PROPERTY IdentifiedBTN : STRING
GET
IF ipMoverTcIo <> 0 THEN
	_IdentifiedBTN := ipMoverTcIo.GetIdentifiedMoverBtn();
END_IF

IdentifiedBTN := _IdentifiedBTN;
END_GET
SET
_IdentifiedBTN := IdentifiedBTN;
END_SET
END_PROPERTY

PROPERTY InStation : BOOL
GET
InStation := _InStation;
END_GET
SET
_InStation := InStation;
END_SET
END_PROPERTY

METHOD LeaveMovementArea : I_PlanarTaskResult
LeaveMovementArea := LeaveMvmtAreaTask.Execute();
END_METHOD

PROPERTY MoveCommand : I_MoveCommands
GET
MoveCommand := THIS^;
END_GET
END_PROPERTY

PROPERTY MoverBTN : STRING
GET
IF ipMoverTcIo <> 0 THEN
	_MoverBTN := ipMoverTcIo.GetBtn();
END_IF

MoverBTN := _MoverBTN;
END_GET
END_PROPERTY

PROPERTY MoverIndex : UDINT
GET
MoverIndex := _MoverIndex;
END_GET
SET
_MoverIndex := MoverIndex;
END_SET
END_PROPERTY

PROPERTY MoverType : XPlanarMoverType
GET
MoverType := _MoverType;
END_GET
SET
_MoverType := MoverType;
END_SET
END_PROPERTY

PROPERTY ObjectInfo : REFERENCE TO PlanarObjectInfo
GET
ObjectInfo ref= _ObjectInfo;
END_GET
END_PROPERTY

{attribute 'suppress_wrn_C0410'}
PROPERTY pm : REFERENCE TO MC_PlanarMover
GET
pm ref= _Mover;
END_GET
END_PROPERTY

METHOD PUBLIC Reset : I_PlanarTaskResult
Reset := ResetMover.Execute();
END_METHOD

PROPERTY RotationModulo : LREAL
GET
RotationModulo := _ModuloPosC;
END_GET
END_PROPERTY

{attribute 'suppress_wrn_C0410'}
PROPERTY Status : REFERENCE TO CDT_MCTOPLC_PLANAR_MOVER_STD
GET
Status ref= _Std;
END_GET
END_PROPERTY

PROPERTY Utility : I_TcIoXPlanarMover
GET
IF ipMoverTcIo <> 0 THEN
	Utility := ipMoverTcIo;
END_IF
END_GET
SET
ipMoverTcIo := Utility;
END_SET
END_PROPERTY

METHOD CyclicLogic
VAR
	Result : BOOL;
END_VAR

VAR_INST
	MoverSetPos	 : MoverVector;
	SetPosX		 : LREAL;
	SetPosY		 : LREAL;
	ModXPos		 : LREAL;
	ModXPosRound : LREAL;
	ModYPos		 : LREAL;
	ModYPosRound : LREAL;
	FracX		 : LREAL;
	FracY		 : LREAL;
END_VAR
//Keep Task command feedbacks up to date
EnableMover.CyclicLogic();
DisableMover.CyclicLogic();
HaltMover.CyclicLogic();
JoinMoverToTrack.CyclicLogic();
LeaveMoverFromTrack.CyclicLogic();
ResetMover.CyclicLogic();
MoveOnTrackXY.CyclicLogic();
MoveOnTrack.CyclicLogic();
RotateMover.CyclicLogic();
XMove.CyclicLogic();
YMove.CyclicLogic();
ZMove.CyclicLogic();
AMove.CyclicLogic();
BMove.CyclicLogic();
XMoveRelative.CyclicLogic();
YMoveRelative.CyclicLogic();
CMoveRelative.CyclicLogic();
XMoveVelocity.CyclicLogic();
YMoveVelocity.CyclicLogic();
CMoveVelocity.CyclicLogic();
MoveToPosition.CyclicLogic();
AddMoverToGroup.CyclicLogic();
JoinToClosestTrack.CyclicLogic();
SquareMover.CyclicLogic();
RunExternalSetpointRelativeMode.CyclicLogic();
StopExternalSetpoint.CyclicLogic();
EnterMvmtAreaTask.CyclicLogic();
LeaveMvmtAreaTask.CyclicLogic();

IF NOT _Initialized THEN
	RETURN;
END_IF

//Update Mover MC Info
_std	 := _Mover.MCTOPLC.STD;
_Busy	 := _std.Busy.busyMover;
_Error	 := _Mover.Error;
_ErrorID := _Mover.ErrorId;

//Get Current Mover Position
_PreviousActPos := _MoverActPos;
_MoverActPos := _Mover.MCTOPLC.ACT.ActPos;

//Calculate Mover Closest Quarter Angle
_ModuloPosC	 := MODABS(_MoverActPos.c, 360.0);
IF _ModuloPosC < 315.0 AND _ModuloPosC > 225.0 THEN
	_ClosestQuarterAngle := 270.0;
ELSIF _ModuloPosC < 225.0 AND _ModuloPosC > 135.0 THEN
	_ClosestQuarterAngle := 180.0;
ELSIF _ModuloPosC < 135.0 AND _ModuloPosC > 45.0 THEN
	_ClosestQuarterAngle := 90.0;
ELSE
	_ClosestQuarterAngle := 0.0;
END_IF

//Determine if Mover is at a valid rotation position
MoverSetPos			:= _Mover.MCTOPLC.SET.SetPos;
SetPosX				:= TO_LREAL(TO_DINT(MoverSetPos.x * (2 * 10))) / (2 * 10); //Round the X position to 2 decimal places
SetPosY				:= TO_LREAL(TO_DINT(MoverSetPos.y * (2 * 10))) / (2 * 10); //Round the X position to 2 decimal places
ModXPos				:= LMOD(MoverSetPos.x, XPlanar.RotationMultiplier);
ModXPosRound		:= TO_LREAL(TO_DINT(ModXPos * (2 * 10))) / (2 * 10); //Round the Modulo position to 2 decimal places
FracX				:= FRAC(ModXPosRound);
ModYPos				:= LMOD(MoverSetPos.y, XPlanar.RotationMultiplier);
ModYPosRound		:= TO_LREAL(TO_DINT(ModYPos * (2 * 10))) / (2 * 10); //Round the Modulo position to 2 decimal places
FracY				:= FRAC(ModYPosRound);

//If APS42xx tiles are detected allow rotation anywhere on driver version 5 and above
IF Tc3_XPlanarUtility.Global_Version.stLibVersion_Tc3_XPlanarUtility.iMajor >= 5 AND XPlanar.RotationMultiplier = 80  THEN
	_AtRotationPosition := TRUE;
ELSE
	_AtRotationPosition := (SetPosX >= (XPlanar.RotationMultiplier - 0.25) AND FracX = 0) AND (SetPosY >= (XPlanar.RotationMultiplier - 0.25) AND FracY = 0);
END_IF

//Monitor Changes in move dynamic settings
IF UpdateMoveDynamics THEN
	_DynMove.SetValuesVADJ(_MoveDynamics.Velocity,
						   _MoveDynamics.Accel,
						   _MoveDynamics.Decel,
						   _MoveDynamics.Jerk);

	_DynTrackMove.SetValuesVADJ(_MoveDynamics.Velocity,
								_MoveDynamics.Accel,
								_MoveDynamics.Decel,
								_MoveDynamics.Jerk);

	UpdateMoveDynamics := FALSE;
END_IF

IF UpdateRotateDynamics THEN
	_DynRotate.SetLimit(Coord_Mcs_C1,
						_RotateDynamics.Velocity,
						_RotateDynamics.Accel,
						_RotateDynamics.Decel,
						_RotateDynamics.Jerk);

	UpdateRotateDynamics := FALSE;
END_IF

IF UpdateTiltDynamics THEN
	_DynRotate.SetLimit(Coord_Mcs_A1,
						_TiltDynamics.Velocity,
						_TiltDynamics.Accel,
						_TiltDynamics.Decel,
						_TiltDynamics.Jerk);

	_DynRotate.SetLimit(Coord_Mcs_B1,
						_TiltDynamics.Velocity,
						_TiltDynamics.Accel,
						_TiltDynamics.Decel,
						_TiltDynamics.Jerk);

	UpdateTiltDynamics := FALSE;
END_IF

//Update Mover Position for HMI
IF _MoverIndex > 0 AND _MoverIndex <= HmiObjectCounts.Movers THEN
	XPlanarHMI.MoverPositions[_MoverIndex]		  := _MoverActPos;
	XPlanarHMI.MoverObjects[_MoverIndex].MoverBTN := _MoverBTN;
	XPlanarHMI.MoverObjects[_MoverIndex].Error	  := _Error;
END_IF
END_METHOD

//FB_Init is always available implicitly and it is used primarily for initialization.
//The return value is not evaluated. For a specific influence, you can also declare the
//methods explicitly and provide additional code there with the standard initialization
//code. You can evaluate the return value.
METHOD FB_Init: BOOL
VAR_INPUT
    bInitRetains: BOOL; // TRUE: the retain variables are initialized (reset warm / reset cold)
    bInCopyCode: BOOL;  // TRUE: the instance will be copied to the copy code afterward (online change)   
END_VAR
VAR
	i	: UINT;
END_VAR
IF NOT bInCopyCode THEN
	FOR i := 1 TO Tc3_XPlanarUtility.Param_TcIoXPlanarEnvironment.MaxMcPlanarMovers DO
		IF ip.Movers[i] = 0 THEN
			ip.Movers[i] := THIS^;
			ip.Movers[i].MoverIndex := i;
			EXIT;
		END_IF 
	END_FOR
END_IF
END_METHOD

PROPERTY LastCyclePosition : Reference TO MoverVector
GET
LastCyclePosition ref= _PreviousActPos;
END_GET
END_PROPERTY

PROPERTY MoverData : I_MoverData
GET
MoverData := _MoverData;
END_GET
SET
_MoverData := MoverData;
END_SET
END_PROPERTY

END_FUNCTION_BLOCK

// Part/Tasks/FB_AllowEnable
FUNCTION_BLOCK FB_AllowEnable EXTENDS FB_PartTask
VAR
END_VAR

METHOD Execute : I_PlanarTaskResult
VAR_INPUT
END_VAR
IF NOT HasRun THEN
	_Done	 := FALSE;
	_Error	 := FALSE;
	_Busy	 := FALSE;
	_ErrorID := 0;
	ipPart.pm.AllowEnable(_PlanarFb);
	HasRun := TRUE;
END_IF

Execute := THIS^;

//Heartbeat that the method is active
ExecuteWatchdog := ExecuteWatchdog + 1;
END_METHOD

END_FUNCTION_BLOCK

// Part/Tasks/FB_ForceDisable
FUNCTION_BLOCK FB_ForceDisable EXTENDS FB_PartTask
VAR
END_VAR

METHOD Execute : I_PlanarTaskResult
VAR_INPUT
END_VAR
IF NOT HasRun THEN
	_Done	 := FALSE;
	_Error	 := FALSE;
	_Busy	 := FALSE;
	_ErrorID := 0;
	ipPart.pm.ForceDisable(_PlanarFb);
	HasRun := TRUE;
END_IF

Execute := THIS^;

//Heartbeat that the method is active
ExecuteWatchdog := ExecuteWatchdog + 1;
END_METHOD

END_FUNCTION_BLOCK

// Part/Tasks/FB_Initialize
FUNCTION_BLOCK FB_Initialize EXTENDS FB_PartTask
VAR
END_VAR

METHOD Execute : I_PlanarTaskResult
VAR_INPUT
	OID : OTCID;
END_VAR
IF NOT HasRun THEN
	ipPart.pm.Initialize(_PlanarFb, OID, XPlanar.Environment);
	HasRun := TRUE;
END_IF

Execute := THIS^;

//Heartbeat that the method is active
ExecuteWatchdog := ExecuteWatchdog + 1;
END_METHOD

END_FUNCTION_BLOCK

// Part/Tasks/FB_ResetPart
FUNCTION_BLOCK FB_ResetPart EXTENDS FB_PartTask
VAR
END_VAR

METHOD Execute : I_PlanarTaskResult
VAR_INPUT
END_VAR
IF NOT HasRun THEN
	_Done	 := FALSE;
	_Error	 := FALSE;
	_Busy	 := FALSE;
	_ErrorID := 0;
	ipPart.pm.Reset(_PlanarFb);
	HasRun := TRUE;
END_IF

Execute := THIS^;

//Heartbeat that the method is active
ExecuteWatchdog := ExecuteWatchdog + 1;
END_METHOD

END_FUNCTION_BLOCK

// Part/FB_XPlanarPart
{attribute 'no_assign'}
{attribute 'no_explicit_call' := 'do not call this POU directly'}
FUNCTION_BLOCK FB_XPlanarPart IMPLEMENTS I_XPlanarPart
VAR
	{attribute 'suppress_wrn_C0540'}
	PlanarPart			 : MC_PlanarPart;
	_Busy				 : BOOL;
	_Error				 : BOOL;
	_ErrorID			 : UDINT;
	_ObjectID			 : OTCID;
	InitPart			 : FB_Initialize   := (Part := THIS^);
	AllowPartEnable		 : FB_AllowEnable  := (Part := THIS^);
	ForcePartDisable	 : FB_ForceDisable := (Part := THIS^);
	ResetPart			 : FB_ResetPart	   := (Part := THIS^);
	InvalidCommandResult : FB_TaskResult   := (Busy := FALSE, Error := TRUE, ErrorID := 9999);
END_VAR

PROPERTY Busy : BOOL
GET
Busy := _Busy;
END_GET
END_PROPERTY

METHOD PUBLIC CyclicLogic
VAR_INPUT
END_VAR
InitPart.CyclicLogic();
AllowPartEnable.CyclicLogic();
ForcePartDisable.CyclicLogic();
ResetPart.CyclicLogic();
END_METHOD

PROPERTY Error : BOOL
GET
Error := _Error;
END_GET
END_PROPERTY

PROPERTY ErrorId : UDINT
GET
ErrorId := ErrorID;
END_GET
END_PROPERTY

METHOD ForceDisable : I_PlanarTaskResult
ForceDisable := ForcePartDisable.Execute();
END_METHOD

METHOD Initialize : I_PlanarTaskResult
VAR_INPUT
END_VAR
IF _ObjectID <> 0 THEN
	Initialize := InitPart.Execute(_ObjectID);
ELSE
	Initialize := InvalidCommandResult;
END_IF
END_METHOD

PROPERTY ObjectID : OTCID
GET
ObjectID := _ObjectID;
END_GET
SET
_ObjectID := ObjectID;
END_SET
END_PROPERTY

{attribute 'suppress_wrn_C0410'}
PROPERTY pm : REFERENCE TO MC_PlanarPart
GET
pm  ref= PlanarPart;
END_GET
END_PROPERTY

METHOD Reset : I_PlanarTaskResult
VAR_INPUT
END_VAR
Reset := ResetPart.Execute();
END_METHOD

METHOD SetAllowEnable : I_PlanarTaskResult
SetAllowEnable := AllowPartEnable.Execute();
END_METHOD

{attribute 'suppress_wrn_C0410'}
PROPERTY State : REFERENCE TO MC_PLANAR_STATE
GET
State := PlanarPart.State;
END_GET
END_PROPERTY

END_FUNCTION_BLOCK

// PositionTrigger/FB_XPlanarPositionTrigger
FUNCTION_BLOCK FB_XPlanarPositionTrigger IMPLEMENTS I_Cyclic, I_XPlanarPositionTrigger
VAR
	_Position		  : FB_PositionXY;
	_Queue			  : FB_MoverQueue;
	_RegisteredMovers : FB_MoverList;
	AllMovers		  : BOOL;
END_VAR

METHOD CyclicLogic
WatchForMover();
END_METHOD

METHOD DeregisterMover
VAR_INPUT
	Mover	: I_XPlanarMover;
END_VAR
_RegisteredMovers.RemoveMover(Mover);
END_METHOD

METHOD GetMover : I_XPlanarMover
GetMover := _Queue.Dequeue();
END_METHOD

PROPERTY MoverIsPresent : BOOL
GET
MoverIsPresent := _Queue.Count > 0;
END_GET
END_PROPERTY

PROPERTY MoverQueue : I_MoverQueue
GET
MoverQueue := _Queue;
END_GET
END_PROPERTY

PROPERTY Position : I_HasPosition
GET
Position := _Position;
END_GET
END_PROPERTY

METHOD RegisterAllMovers
AllMovers := TRUE;
END_METHOD

METHOD RegisterMover
VAR_INPUT
	Mover	: I_XPlanarMover;
END_VAR
VAR
	i : UDINT;
END_VAR
FOR i := 1 TO _RegisteredMovers.Count DO
	IF _RegisteredMovers.List[i] = Mover THEN
		RETURN;
	END_IF
END_FOR
_RegisteredMovers.AddMover(Mover);
END_METHOD

METHOD WatchForMover
VAR_INST
	i : UDINT;
END_VAR

VAR
	idx: UDINT;
END_VAR
IF AllMovers THEN
	FOR i := 1 TO XPlanar.MoverCount DO
		IF ip.Movers[i] <> 0 AND_THEN _Position.x > 0 AND _Position.y > 0 THEN
			IF (ip.Movers[i].ActualPosition.x >= _Position.x - 10 AND ip.Movers[i].ActualPosition.x <= _Position.x + 10) THEN 		//Paint the window in X
				IF _Position.y >= ip.Movers[i].LastCyclePosition.y AND _Position.y <= ip.Movers[i].ActualPosition.y OR 				//Wach for threshold in Y	
					_Position.y <= ip.Movers[i].LastCyclePosition.y AND _Position.y >= ip.Movers[i].ActualPosition.y THEN
						_Queue.Enqueue(ip.Movers[i]);
				END_IF
			ELSIF (ip.Movers[i].ActualPosition.y >= _Position.y - 10 AND ip.Movers[i].ActualPosition.y <= _Position.y + 10) THEN	//Paint the window in Y
				IF _Position.x >= ip.Movers[i].LastCyclePosition.x AND _Position.x <= ip.Movers[i].ActualPosition.x OR				//Wach for threshold in X
					_Position.x <= ip.Movers[i].LastCyclePosition.x AND _Position.x >= ip.Movers[i].ActualPosition.x THEN
						_Queue.Enqueue(ip.Movers[i]);
				END_IF
			END_IF
		END_IF
	END_FOR
ELSE
	FOR i := 1 TO _RegisteredMovers.Count DO
		IF _RegisteredMovers.List[i] <> 0 AND_THEN _Position.x > 0 AND _Position.y > 0 THEN
			IF (_RegisteredMovers.List[i].ActualPosition.x >= _Position.x - 10 AND _RegisteredMovers.List[i].ActualPosition.x <= _Position.x + 10) THEN 		//Paint the window in X
				IF _Position.y >= _RegisteredMovers.List[i].LastCyclePosition.y AND _Position.y <= _RegisteredMovers.List[i].ActualPosition.y OR 				//Wach for threshold in Y	
					_Position.y <= _RegisteredMovers.List[i].LastCyclePosition.y AND _Position.y >= _RegisteredMovers.List[i].ActualPosition.y THEN
						_Queue.Enqueue(_RegisteredMovers.List[i]);
				END_IF
			ELSIF (_RegisteredMovers.List[i].ActualPosition.y >= _Position.y - 10 AND _RegisteredMovers.List[i].ActualPosition.y <= _Position.y + 10) THEN		//Paint the window in Y
				IF _Position.x >= _RegisteredMovers.List[i].LastCyclePosition.x AND _Position.x <= _RegisteredMovers.List[i].ActualPosition.x OR				//Wach for threshold in X
					_Position.x <= _RegisteredMovers.List[i].LastCyclePosition.x AND _Position.x >= _RegisteredMovers.List[i].ActualPosition.x THEN
						_Queue.Enqueue(_RegisteredMovers.List[i]);
				END_IF
			END_IF
		END_IF
	END_FOR	
END_IF
END_METHOD

END_FUNCTION_BLOCK

// PositionTrigger/I_XPlanarPositionTrigger
INTERFACE I_XPlanarPositionTrigger EXTENDS I_Cyclic

METHOD DeregisterMover
VAR_INPUT
	Mover	: I_XPlanarMover;
END_VAR
END_METHOD

METHOD GetMover : I_XPlanarMover
END_METHOD

PROPERTY MoverIsPresent : BOOL
GET
END_GET
END_PROPERTY

PROPERTY MoverQueue : I_MoverQueue
GET
END_GET
END_PROPERTY

PROPERTY Position : I_HasPosition
GET
END_GET
END_PROPERTY

METHOD RegisterAllMovers
END_METHOD

METHOD RegisterMover
VAR_INPUT
	Mover	: I_XPlanarMover;
END_VAR
END_METHOD

END_INTERFACE

// Project Information/F_GetCompany
// This function has been automatically generated from the project information.
{attribute 'signature_flag' := '1073741824'}
{attribute 'TcGenerated'}
{attribute 'no-analysis'}
FUNCTION F_GetCompany : WSTRING
VAR_INPUT
	
END_VAR

F_GetCompany := "Beckhoff Automation LLC";

END_FUNCTION

// Project Information/F_GetTitle
// This function has been automatically generated from the project information.
{attribute 'signature_flag' := '1073741824'}
{attribute 'TcGenerated'}
{attribute 'no-analysis'}
FUNCTION F_GetTitle : WSTRING
VAR_INPUT
	
END_VAR

F_GetTitle := "XPlanarApplication";

END_FUNCTION

// Project Information/F_GetVersion
// This function has been automatically generated from the project information.
{attribute 'signature_flag' := '1073741824'}
{attribute 'TcGenerated'}
{attribute 'no-analysis'}
FUNCTION F_GetVersion : ST_LibVersion
VAR_INPUT
	
END_VAR

F_GetVersion.iMajor := 2;
F_GetVersion.iMinor := 0;
F_GetVersion.iBuild := 6;
F_GetVersion.iRevision := 0;
F_GetVersion.sVersion := '2.0.6';
F_GetVersion.nFlags := 0;

END_FUNCTION

// Station/FB_XPlanarStationBase
{attribute 'no_assign_warning'}
{attribute 'no_explicit_call' := 'do not call this POU directly'}
FUNCTION_BLOCK FB_XPlanarStationBase IMPLEMENTS I_Cyclic, I_XPlanarStation
VAR
	_Name				 : STRING;
	_Busy				 : BOOL;
	_Error				 : BOOL;
	_ErrorID			 : UDINT;
	_Position			 : PositionXYC; //Position of center of the zone
	ipCurrentMover		 : I_XPlanarMover;
	_MoverList			 : FB_MoverList;
	_NumMoversRequired	 : UDINT := 1;
	_ID					 : UDINT;
	_Size				 : Position2D_LREAL := (x := 50, y := 50); //Size of station in mm
	_HasMover			 : BOOL;
	_Occupied			 : BOOL;
	ipTrackID			 : UDINT;		 //ID of track that zone resides on
	_CanReleaseMover	 : BOOL := TRUE; //Set to 0 if station area is blocked
	_StationReady AT %Q* : BOOL;
	ipNextStation		 : I_XPlanarStation;
	_AllowQueing		 : BOOL := TRUE;
	_StationComplete	 : BOOL;
	_StationType		 : E_StationType := E_StationType.Process;
	PrepState			 : UDINT;
	StationState		 : E_XplanarStationState;
	i					 : UDINT := 1;
	CommandResult		 : I_PlanarTaskResult;
	_Process			 : I_StationProcess;
END_VAR

PROPERTY Process : I_StationProcess
GET
IF _Process <> 0 THEN
	Process := _Process;
END_IF
END_GET
SET
_Process := Process;
END_SET
END_PROPERTY

PROPERTY AllowQueing : BOOL
GET
AllowQueing := _AllowQueing;
END_GET
SET
_AllowQueing := AllowQueing;
END_SET
END_PROPERTY

PROPERTY CanReleaseMover : BOOL
SET
_CanReleaseMover := CanReleaseMover;
END_SET
END_PROPERTY

PROPERTY CurrentMover : I_XPlanarMover
GET
IF ipCurrentMover <> 0 THEN
	CurrentMover := ipCurrentMover;
END_IF
END_GET
END_PROPERTY

PROPERTY Error : BOOL
GET
Error := _Error;
END_GET
END_PROPERTY

METHOD Execute
WatchForMover();
IF ipCurrentMover <> 0 THEN
	CASE StationState OF
		E_XplanarStationState.StationIdle: //Wait for mover to arrive in position
			IF _HasMover AND _StationReady AND NOT _StationComplete THEN
				IF ipCurrentMover <> 0 THEN
					IF (ipTrackID <> 0 AND (ipCurrentMover.Status.CommandMode = MC_PLANAR_MOVER_COMMAND_MODE.OnTrack OR ipCurrentMover.Status.CommandMode = MC_PLANAR_MOVER_COMMAND_MODE.CRotationOnTrack)) OR (ipTrackID = 0 AND (ipCurrentMover.Status.CommandMode = MC_PLANAR_MOVER_COMMAND_MODE.FreeMovement OR ipCurrentMover.Status.CommandMode = MC_PLANAR_MOVER_COMMAND_MODE.CRotationFreeMovement))
						THEN
						StationState := E_XplanarStationState.ProcessMover;
					END_IF
				END_IF
			END_IF

		E_XplanarStationState.ProcessMover: //Perform the desired processes with the mover
			IF _Process <> 0 AND_THEN _Process.Execute(ipCurrentMover) THEN
				StationState := E_XplanarStationState.SquareUpMover;
			ELSIF _StationComplete THEN
				StationState := E_XplanarStationState.SquareUpMover;
			END_IF

		E_XplanarStationState.SquareUpMover: //Check mover for angle that allows X/Y Movement
			IF (ipCurrentMover.Status.CommandMode = MC_PLANAR_MOVER_COMMAND_MODE.CRotationOnTrack) OR (ipCurrentMover.Status.CommandMode = MC_PLANAR_MOVER_COMMAND_MODE.CRotationFreeMovement) THEN
				CommandResult := ipCurrentMover.MoveCommand.SquareUp();
				IF CommandResult.Done THEN
					StationState := E_XplanarStationState.SendMoverAway;
				END_IF
			ELSE
				StationState := E_XplanarStationState.SendMoverAway;
			END_IF

		E_XplanarStationState.SendMoverAway: //Send the current lead mover away
			IF ipNextStation <> 0 AND _CanReleaseMover THEN
				IF (NOT ipNextStation.HasMover OR ipNextStation.AllowQueing) THEN
					CommandResult := ipCurrentMover.MoveCommand.SendToStation(Destination := ipNextStation);
					IF CommandResult.Busy THEN
						StationState := E_XplanarStationState.CycleComplete;
					END_IF
				END_IF
			END_IF

		E_XplanarStationState.CycleComplete: //Mover on its way out
			_StationReady := FALSE;
			StationState  := E_XplanarStationState.StationIdle;

		E_XPlanarStationState.StationError:
			_Error := TRUE;
	END_CASE
ELSE
	_StationComplete := FALSE;
	_StationReady	 := FALSE;
	StationState	 := E_XplanarStationState.StationIdle;
END_IF
END_METHOD

PROPERTY HasMover : BOOL
GET
HasMover := _HasMover;
END_GET
SET
_HasMover := HasMover;
END_SET
END_PROPERTY

PROPERTY ID : UDINT
GET
ID := _ID;
END_GET
SET
_ID := ID;
END_SET
END_PROPERTY

{attribute 'suppress_wrn_C0410'}
PROPERTY MoverList : REFERENCE TO FB_MoverList
GET
MoverList ref= _MoverList;
END_GET
END_PROPERTY

PROPERTY NextStation : I_XPlanarStation
GET
NextStation := ipNextStation;
END_GET
SET
ipNextStation := NextStation;
END_SET
END_PROPERTY

{attribute 'suppress_wrn_C0410'}
PROPERTY Position : REFERENCE TO PositionXYC
GET
Position ref= _Position;
END_GET
END_PROPERTY

METHOD Reset : BOOL
StationState := E_XplanarStationState.StationIdle;
PrepState	 := 0;
_Error		 := FALSE;
Reset		 := true;
END_METHOD

{attribute 'suppress_wrn_C0410'}
PROPERTY Size : REFERENCE TO Position2D_LREAL
GET
Size ref= _Size;
END_GET
END_PROPERTY

PROPERTY StationComplete : BOOL
SET
_StationComplete := StationComplete;
END_SET
END_PROPERTY

PROPERTY StationReady : BOOL
GET
StationReady := _StationReady;
END_GET
END_PROPERTY

PROPERTY StationType : E_StationType
GET
StationType := _StationType;
END_GET
SET
_StationType := StationType;
END_SET
END_PROPERTY

PROPERTY TrackID : UDINT
GET
TrackID := ipTrackID;
END_GET
SET
ipTrackID := TrackID;
END_SET
END_PROPERTY

METHOD CyclicLogic
VAR
	i : UDINT;
END_VAR
IF _ID > 0 AND _ID <= XPlanar.StationCount THEN
	XPlanarHMI.StationObjects[_ID].Width  := TO_DINT(_Size.x);
	XPlanarHMI.StationObjects[_ID].Height := TO_DINT(_Size.y);
	XPlanarHMI.StationObjects[_ID].X	  := TO_DINT(_Position.x);
	XPlanarHMI.StationObjects[_ID].Y	  := TO_DINT(_Position.y);
END_IF

_Busy := _HasMover;

//Create a queue of all movers destined for this station
_MoverList.Clear();
FOR i := 1 TO XPlanar.MoverCount DO
	IF ip.Movers[i] <> 0 AND ip.Movers[i].Destination <> 0 THEN
		IF ip.Movers[i].Destination.ID = _ID THEN
			_MoverList.AddMover(ip.Movers[i]);
		END_IF
	END_IF
END_FOR
END_METHOD

//FB_Init is always available implicitly and it is used primarily for initialization.

//The return value is not evaluated. For a specific influence, you can also declare the

//methods explicitly and provide additional code there with the standard initialization

//code. You can evaluate the return value.
METHOD FB_Init : BOOL
VAR_INPUT
	bInitRetains : BOOL; // TRUE: the retain variables are initialized (reset warm / reset cold)
	bInCopyCode	 : BOOL; // TRUE: the instance will be copied to the copy code afterward (online change)   
END_VAR

VAR
	i : UINT;
END_VAR
IF NOT bInCopyCode THEN
	FOR i := 1 TO SystemParameters.MAX_STATION_COUNT DO
		IF ip.Stations[i] = 0 THEN
			ip.Stations[i] := THIS^;
			ip.Stations[i].ID := i;
			XPlanar.StationCount := i;
			EXIT;
		END_IF
	END_FOR
END_IF
END_METHOD

PROPERTY Name : STRING
GET
Name := _Name;
END_GET
SET
_Name := Name;
END_SET
END_PROPERTY

METHOD WatchForMover
VAR_INST
	idx : UDINT;
END_VAR
FOR idx := 1 TO XPlanar.MoverCount DO
	IF ip.Movers[idx] <> 0 THEN
		IF _Position.x > 0 AND _Position.y > 0 THEN
			IF (ip.Movers[idx].ActualPosition.x + 50 >= _Position.x - (_Size.x / 2) AND ip.Movers[idx].ActualPosition.x - 50 <= _Position.x + (_Size.x / 2)) AND
			   (ip.Movers[idx].ActualPosition.y + 50 >= _Position.y - (_Size.y / 2) AND ip.Movers[idx].ActualPosition.y - 50 <= _Position.y + (_Size.y / 2)) THEN
				IF ip.Movers[idx].Destination <> 0 THEN
					IF ip.Movers[idx].Destination.ID = _ID THEN
						ipCurrentMover := ip.Movers[idx];
						_HasMover := TRUE;
						EXIT;
					ELSE
						ipCurrentMover := 0;
						_HasMover := FALSE;
					END_IF
				END_IF
			END_IF
		END_IF
	END_IF
END_FOR

IF _HasMover AND ipCurrentMover <> 0 THEN
	IF ipCurrentMover <> 0 THEN
		CASE _StationType OF
			E_StationType.Process:
				_StationReady := NOT ipCurrentMover.Status.Busy.busyMover;

			E_StationType.DecisionPoint:
				_StationReady := _HasMover;
		END_CASE
	END_IF
END_IF
END_METHOD

END_FUNCTION_BLOCK

// Tile/FB_XPlanarTile
{attribute 'no_assign'}
{attribute 'no_explicit_call' := 'do not call this POU directly'}
FUNCTION_BLOCK FB_XPlanarTile
VAR
	_Busy				: BOOL;
	_Error				: BOOL;
	_ErrorID			: UDINT;
	_Utility			: I_TcIoXPlanarTile;
	_Index				: UINT;
	_Part				: UINT := 1;
	_Btn				: STRING(13);
	_DcLinkVoltage		: UINT;
	_DcLinkOk			: BOOL;
	_TimeToShutdown		: LREAL;
	_ObservedPower		: LREAL;
	_OverLimitFactor	: LREAL;
	_DiagData			: POINTER TO ST_CoeDriveDiagData;
	_Position			: ST_TcIoTilePositionOnPart;
	_Temperatures		: ST_TileTemperatures;
	_TileType			: TileType;
	CoEUpdateTimer		: TON;
	CriticalUpdateTimer : TON;
	DiagDataResult		: ULINT;
END_VAR

PROPERTY Btn : STRING(13)
GET
Btn := _Btn;
END_GET
END_PROPERTY

PROPERTY Busy : BOOL
GET
Busy := _Busy;
END_GET
END_PROPERTY

METHOD PUBLIC CyclicLogic
VAR_INST
	UpdateTileData : BOOL;
	test   : DINT;
END_VAR
(*IF XPlanar.OperationMode = Tc3_XPlanarUtility.XPlanarOperationMode.Normal THEN
	IF SystemParameters.TileDiagUpdate > 0 THEN
		CoEUpdateTimer(IN := NOT UpdateTileData, PT := TO_TIME(SystemParameters.TileDiagUpdate) * 1000);
		IF CoEUpdateTimer.Q THEN
			UpdateTileData := TRUE;
		END_IF

		test := SIZEOF(_diagdata);

		//Update the tile diagnostic data
		IF UpdateTileData AND_THEN XPlanar.EnvironmentTcIo.TcIoXpu(1).TcIoTile(_Part, Index).CoE.DiagData.Update() THEN
			_DiagData := XPlanar.EnvironmentTcIo.TcIoXpu(1).TcIoTile(_Part, Index).CoE.DiagData.All;
			_DcLinkOk := XPlanar.EnvironmentTcIo.TcIoXpu(1).TcIoTile(_Part, Index).CoE.DiagData.DcLinkOk;
			UpdateTileData	  := FALSE;
		END_IF

		CriticalUpdateTimer(IN := NOT CriticalUpdateTimer.Q, PT := T#1S);
		IF CriticalUpdateTimer.Q THEN
			_TimeToShutdown	 := XPlanar.EnvironmentTcIo.TcIoXpu(1).TcIoTile(_Part, Index).GetTimeToShutdown();
			_ObservedPower	 := XPlanar.EnvironmentTcIo.TcIoXpu(1).TcIoTile(_Part, Index).GetObservedTilePower();
			_OverLimitFactor := XPlanar.EnvironmentTcIo.TcIoXpu(1).TcIoTile(_Part, Index).GetPowerOverLimitFactor();
		END_IF
	ELSE
		UpdateTileData := FALSE;
	END_IF
END_IF
*)
END_METHOD

PROPERTY DcLinkOk : BOOL
GET
DcLinkOk := _DcLinkOk;
END_GET
END_PROPERTY

PROPERTY Error : BOOL
GET
Error := _Error;
END_GET
END_PROPERTY

PROPERTY ErrorId : UDINT
GET
ErrorId := ErrorID;
END_GET
END_PROPERTY

PROPERTY Index : UINT
GET
Index := _Index;
END_GET
SET
_Index := Index;
END_SET
END_PROPERTY

METHOD Initialize : BOOL
//Get the Tile Type
_TileType := XPlanar.EnvironmentTcIo.TcIoXpu(1).TcIoTile(_Part, _Index).GetTileType();

//Get the configured position of the tile
_Position := XPlanar.EnvironmentTcIo.TcIoXpu(1).TcIoTile(_Part, _Index).TilePositionOnPart();

//Get BTN of tile
_Btn := XPlanar.EnvironmentTcIo.TcIoXpu(1).TcIoTile(_Part, _Index).GetBtn();

//Update the object array for HMI
IF _Index > 0 AND _Index <= HMIObjectCounts.Tiles THEN
	//Populate tile position
	XPlanarHMI.TileObjects[_Index].X := TO_DINT(_Position.X);
	XPlanarHMI.TileObjects[_Index].Y := TO_DINT(_Position.Y);
	//Populate tile type
	CASE _TileType OF
		TileType.APS4224_1000_0000:
			XPlanarHMI.TileObjects[_Index].Width  := 160;
			XPlanarHMI.TileObjects[_Index].Height := 320;
			XPlanar.RotationMultiplier			  := 80.0;	
	
		TileType.APS4242_1000_0000:
			XPlanarHMI.TileObjects[_Index].Width  := 320;
			XPlanarHMI.TileObjects[_Index].Height := 160;
			XPlanar.RotationMultiplier			  := 80.0;	
			
		TileType.APS4244_1000_0000:
			XPlanarHMI.TileObjects[_Index].Width  := 320;
			XPlanarHMI.TileObjects[_Index].Height := 320;
			XPlanar.RotationMultiplier			  := 80.0;
	
		TileType.APS4322_0000_0000:
			XPlanarHMI.TileObjects[_Index].Width  := 240;
			XPlanarHMI.TileObjects[_Index].Height := 240;
			XPlanar.RotationMultiplier			  := 120.0;
	
// 			//Get initial diagnostic data
// 			IF _Part > 0 AND _Index > 0 THEN
// 				//ipTileTcIo := XPlanar.EnvironmentTcIo.TcIoXpu(1).TcIoTile(_Part, Index).Aps4322;
// 				IF XPlanar.OperationMode = Tc3_XPlanarUtility.XPlanarOperationMode.Normal THEN
// 					IF XPlanar.EnvironmentTcIo.TcIoXpu(1).TcIoTile(_Part, _Index).Aps4322.CoE.DiagData.Update() THEN
// 						_DiagData := XPlanar.EnvironmentTcIo.TcIoXpu(1).TcIoTile(_Part, _Index).Aps4322.CoE.DiagData.All;
// 					END_IF
// 				END_IF
// 			END_IF
	END_CASE
END_IF
Initialize := TRUE;
END_METHOD

PROPERTY PartIndex : UINT
GET
PartIndex := _Part;
END_GET
SET
_Part := PartIndex;
END_SET
END_PROPERTY

{attribute 'suppress_wrn_C0410'}
PROPERTY PositionOnPart : REFERENCE TO ST_TcIoTilePositionOnPart
GET
PositionOnPart ref= _Position;
END_GET
END_PROPERTY

{attribute 'suppress_wrn_C0410'}
PROPERTY Temperatures : REFERENCE TO ST_TileTemperatures
GET
Temperatures ref= _Temperatures;
END_GET
END_PROPERTY

PROPERTY TimeToShutdown : LREAL
GET
TimeToShutdown := _TimeToShutdown;
END_GET
END_PROPERTY

METHOD Update
VAR_INPUT
END_VAR
// XPlanar.EnvironmentTcIo.TcIoXpu(1).TcIoTile(_Part, Index).CoE.DiagData.Update();
// _DiagData		 := XPlanar.EnvironmentTcIo.TcIoXpu(1).TcIoTile(_Part, Index).CoE.DiagData.All;
// _DcLinkOk		 := XPlanar.EnvironmentTcIo.TcIoXpu(1).TcIoTile(_Part, Index).CoE.DiagData.DcLinkOk;
// _TimeToShutdown	 := XPlanar.EnvironmentTcIo.TcIoXpu(1).TcIoTile(_Part, Index).GetTimeToShutdown();
// _ObservedPower	 := XPlanar.EnvironmentTcIo.TcIoXpu(1).TcIoTile(_Part, Index).GetObservedTilePower();
// _OverLimitFactor := XPlanar.EnvironmentTcIo.TcIoXpu(1).TcIoTile(_Part, Index).GetPowerOverLimitFactor();
END_METHOD

PROPERTY Utility : I_TcIoXPlanarTile
GET
IF _Utility <> 0 THEN
	Utility := _Utility;
end_if
END_GET
END_PROPERTY

END_FUNCTION_BLOCK

// Tile/I_XPlanarTile
INTERFACE I_XPlanarTile EXTENDS __SYSTEM.IQueryInterface

PROPERTY Btn : STRING(13)
GET
END_GET
END_PROPERTY

PROPERTY Busy : BOOL
GET
END_GET
END_PROPERTY

PROPERTY DcLinkOk : BOOL
GET
END_GET
END_PROPERTY

PROPERTY Error : BOOL
GET
END_GET
END_PROPERTY

PROPERTY ErrorId : UDINT
GET
END_GET
END_PROPERTY

PROPERTY Index : UINT
GET
END_GET
SET
END_SET
END_PROPERTY

PROPERTY PartIndex : UINT
GET
END_GET
SET
END_SET
END_PROPERTY

{attribute 'suppress_wrn_C0410'}
PROPERTY PositionOnPart : REFERENCE TO ST_TcIoTilePositionOnPart
GET
END_GET
END_PROPERTY

{attribute 'suppress_wrn_C0410'}
PROPERTY Temperatures : REFERENCE TO ST_TileTemperatures
GET
END_GET
END_PROPERTY

PROPERTY TimeToShutdown : UDINT
GET
END_GET
END_PROPERTY

METHOD Update
VAR_INPUT
END_VAR
END_METHOD

PROPERTY Utility : I_TcIoXPlanarTile
GET
END_GET
END_PROPERTY

END_INTERFACE

// Track/TaskClasses/FB_AddTrackToGroup
FUNCTION_BLOCK FB_AddTrackToGroup EXTENDS FB_TrackTask
VAR
END_VAR

METHOD Execute : I_PlanarTaskResult
VAR_INPUT
	refGroup : REFERENCE TO MC_PlanarGroup;
END_VAR
_Done	 := FALSE;
_Error	 := FALSE;
_Busy	 := FALSE;
_ErrorID := 0;
ipTrack.pm.AddToGroup(_PlanarFb, refGroup);
Execute := THIS^;

//Heartbeat that the method is active
ExecuteWatchdog := ExecuteWatchdog + 1;
END_METHOD

END_FUNCTION_BLOCK

// Track/TaskClasses/FB_AppendLine
{attribute 'no_assign_warning'} 
FUNCTION_BLOCK FB_AppendLine EXTENDS FB_TrackTask
VAR
	StartPoint : PositionXYC;
	EndPoint   : PositionXYC;
END_VAR

METHOD Execute : I_PlanarTaskResult
VAR_INPUT
	StartPointX : LREAL;
	StartPointY : LREAL;
	EndPointX	: LREAL;
	EndPointY	: LREAL;
END_VAR
IF NOT HasRun THEN
	_Done	 := FALSE;
	_Error	 := FALSE;
	_Busy	 := FALSE;
	_ErrorID := 0;
	StartPoint.SetValuesXY(StartPointX, StartPointY);
	EndPoint.SetValuesXY(EndPointX, EndPointY);
	ipTrack.pm.AppendLine(_PlanarFb, StartPoint, EndPoint);
	HasRun := TRUE;
END_IF

Execute := THIS^;

//Heartbeat that the method is active
ExecuteWatchdog := ExecuteWatchdog + 1;
END_METHOD

END_FUNCTION_BLOCK

// Track/TaskClasses/FB_AppendPoint
{attribute 'no_assign_warning'}
FUNCTION_BLOCK FB_AppendPoint EXTENDS FB_TrackTask
VAR
	Position : PositionXYC;
END_VAR

METHOD Execute : I_PlanarTaskResult
VAR_INPUT
	XPoint : LREAL;
	YPoint : LREAL;
END_VAR
IF NOT HasRun THEN
	_Done	 := FALSE;
	_Error	 := FALSE;
	_Busy	 := FALSE;
	_ErrorID := 0;
	Position.SetValuesXY(XPoint, YPoint);
	ipTrack.pm.AppendPosition(_PlanarFb, Position);
	HasRun := TRUE;
END_IF

Execute := THIS^;

//Heartbeat that the method is active
ExecuteWatchdog := ExecuteWatchdog + 1;
END_METHOD

END_FUNCTION_BLOCK

// Track/TaskClasses/FB_BuildTrack
FUNCTION_BLOCK FB_BuildTrack EXTENDS FB_TrackTask
VAR
	BuildTrack	: BOOL;
END_VAR

METHOD PUBLIC CyclicLogic
VAR_INST
	WatchdogCheck : UDINT;
	i			  : UDINT := 1;
END_VAR
_PlanarFb.Update();
CASE TaskState OF
	0: //Init
		THIS^._Busy := FALSE;
		IF BuildTrack THEN
			THIS^._Done	   := FALSE;
			THIS^._Error   := FALSE;
			THIS^._ErrorID := 0;
			THIS^._Busy	   := TRUE;
			BuildTrack	   := FALSE;
			i			   := 1;
			TaskState	   := TaskState + 10;
		END_IF

	10: //Set StartFromTrack
		IF ipTrack.Definition.StartFromTrackID > 0 THEN
			ipTrack.pm.StartFromTrack(_PlanarFb, ip.Tracks[ipTrack.Definition.StartFromTrackID].pm);
			TaskState := TaskState + 1;
		ELSE
			TaskState := TaskState + 10;
		END_IF

	11: //Watch Command Feedback
		IF _PlanarFb.Done THEN
			TaskState := 20;
		ELSIF _PlanarFb.Error THEN
			THIS^._Error			  := TRUE;
			THIS^._ErrorID			  := _PlanarFb.ErrorId;
			THIS^._BlockingObjectInfo := _PlanarFb.objectInfo;
			TaskState				  := 0;
		END_IF

	20: //Append Track Objects
		IF ipTrack.Definition.Items[i].StartPoint.x > 0 THEN
			CASE ipTrack.Definition.Items[i].ItemType OF
				Point:
					ipTrack.pm.AppendPosition(_PlanarFb, ipTrack.Definition.Items[i].StartPoint);

				Line:
					IF ipTrack.Definition.Items[i].EndPoint.x > 0 THEN
						ipTrack.pm.AppendLine(_PlanarFb, ipTrack.Definition.Items[i].StartPoint, ipTrack.Definition.Items[i].EndPoint);
					ELSE
						THIS^._Error			  := TRUE;
						THIS^._ErrorID			  := 9999;
						TaskState				  := 0;	
					END_IF					
					
				Circle:
					ipTrack.pm.AppendCircle(_PlanarFb,
									   ipTrack.Definition.Items[i].StartPoint,
									   ipTrack.Definition.Items[i].EndPoint,
									   ipTrack.Definition.Items[i].CenterPoint,
									   ipTrack.Definition.Items[i].CircleClockwise);
			END_CASE

			TaskState := TaskState + 1;
		ELSE
			TaskState := TaskState + 10; //No Object Defined Exit the loop
		END_IF

	21: //Watch Command Feedback
		IF _PlanarFb.Done THEN
			IF i < SystemParameters.MAX_OBJECTS_PER_TRACK THEN
				i		  := i + 1;
				TaskState := 20;
			ELSE
				i		  := 1;
				TaskState := 30;
			END_IF
		ELSIF _PlanarFb.Error THEN
			THIS^._Error			  := TRUE;
			THIS^._ErrorID			  := _PlanarFb.ErrorId;
			THIS^._BlockingObjectInfo := _PlanarFb.objectInfo;
			TaskState				  := 0;
		END_IF

	30: //Set EndAtTrack
		IF ipTrack.Definition.EndAtTrackID > 0 THEN
			ipTrack.pm.EndAtTrack(_PlanarFb, ip.Tracks[ipTrack.Definition.EndAtTrackID].pm);
			TaskState := TaskState + 1;
		ELSIF ipTrack.Definition.CloseLoop THEN
			ipTrack.pm.CloseLoop(_PlanarFb);
			TaskState := TaskState + 1;
		ELSE
			TaskState := TaskState + 10;
		END_IF

	31: //Watch Command Feedback
		IF _PlanarFb.Done THEN
			TaskState := 40;
		ELSIF _PlanarFb.Error THEN
			THIS^._Error			  := TRUE;
			THIS^._ErrorID			  := _PlanarFb.ErrorId;
			THIS^._BlockingObjectInfo := _PlanarFb.objectInfo;
			TaskState				  := 0;
		END_IF

	40: //Build Complete
		THIS^._Done := TRUE;
		TaskState	:= 0;
END_CASE

IF ExecuteWatchdog <> WatchdogCheck THEN
	WatchdogCheck := ExecuteWatchdog;
ELSE
	HasRun			:= FALSE;
	ExecuteWatchdog := 0;
END_IF
END_METHOD

METHOD Execute : I_PlanarTaskResult
IF NOT HasRun THEN
	_Done	   := FALSE;
	_Error	   := FALSE;
	_Busy	   := FALSE;
	_ErrorID   := 0;
	BuildTrack := TRUE;
	HasRun	   := TRUE;
END_IF

Execute := THIS^;

//Heartbeat that the method is active
ExecuteWatchdog := ExecuteWatchdog + 1;
END_METHOD

END_FUNCTION_BLOCK

// Track/TaskClasses/FB_ClearSegment
FUNCTION_BLOCK FB_ClearSegment EXTENDS FB_TrackTask
VAR
END_VAR

METHOD Execute : I_PlanarTaskResult
IF NOT HasRun THEN
	_Done	 := FALSE;
	_Error	 := FALSE;
	_Busy	 := FALSE;
	_ErrorID := 0;
	ipTrack.pm.Clear(_PlanarFb);
	HasRun := TRUE;
END_IF

Execute := THIS^;

//Heartbeat that the method is active
ExecuteWatchdog := ExecuteWatchdog + 1;
END_METHOD

END_FUNCTION_BLOCK

// Track/TaskClasses/FB_CloseLoop
FUNCTION_BLOCK FB_CloseLoop EXTENDS FB_TrackTask
VAR
END_VAR

METHOD Execute : I_PlanarTaskResult
IF NOT HasRun THEN
	_Done	 := FALSE;
	_Error	 := FALSE;
	_Busy	 := FALSE;
	_ErrorID := 0;
	ipTrack.pm.CloseLoop(_PlanarFb);
	HasRun := TRUE;
END_IF

Execute := THIS^;

//Heartbeat that the method is active
ExecuteWatchdog := ExecuteWatchdog + 1;
END_METHOD

END_FUNCTION_BLOCK

// Track/TaskClasses/FB_DisableTrack
FUNCTION_BLOCK FB_DisableTrack EXTENDS FB_TrackTask
VAR
END_VAR

METHOD Execute : I_PlanarTaskResult
VAR_INPUT
END_VAR
IF ipTrack.Status.State = Mc_Planar_State.Enabled THEN
	_Done	 := FALSE;
	_Error	 := FALSE;
	_Busy	 := FALSE;
	_ErrorID := 0;
	ipTrack.pm.Disable(_PlanarFb);
END_IF

Execute := THIS^;

//Heartbeat that the method is active
ExecuteWatchdog := ExecuteWatchdog + 1;
END_METHOD

END_FUNCTION_BLOCK

// Track/TaskClasses/FB_EnableTrack
FUNCTION_BLOCK FB_EnableTrack EXTENDS FB_TrackTask
VAR
END_VAR

METHOD Execute : I_PlanarTaskResult
VAR_INPUT
END_VAR
IF ipTrack.Status.State = Mc_Planar_State.Disabled THEN
	_Done	 := FALSE;
	_Error	 := FALSE;
	_Busy	 := FALSE;
	_ErrorID := 0;
	ipTrack.pm.Enable(_PlanarFb);
END_IF

Execute := THIS^;

//Heartbeat that the method is active
ExecuteWatchdog := ExecuteWatchdog + 1;
END_METHOD

END_FUNCTION_BLOCK

// Track/TaskClasses/FB_SetEndAtTrack
FUNCTION_BLOCK FB_SetEndAtTrack EXTENDS FB_TrackTask
VAR
	Options : ST_EndAtTrackAdvancedOptions;
END_VAR

METHOD Execute : I_PlanarTaskResult
VAR_INPUT
	SegmentID : UDINT;
END_VAR
IF NOT HasRun AND (SegmentID > 0 AND SegmentID <= XPlanar.TrackCount) THEN
	_Done	 := FALSE;
	_Error	 := FALSE;
	_Busy	 := FALSE;
	_ErrorID := 0;
	ipTrack.pm.EndAtTrack(_PlanarFb, ip.Tracks[SegmentID].pm);
	HasRun := TRUE;
END_IF

Execute := THIS^;

//Heartbeat that the method is active
ExecuteWatchdog := ExecuteWatchdog + 1;
END_METHOD

END_FUNCTION_BLOCK

// Track/TaskClasses/FB_SetStartFromTrack
FUNCTION_BLOCK FB_SetStartFromTrack EXTENDS FB_TrackTask
VAR
	Options : ST_StartFromTrackAdvancedOptions;
END_VAR

METHOD Execute : I_PlanarTaskResult
VAR_INPUT
	SegmentID : UDINT;
END_VAR
IF NOT HasRun AND (SegmentID > 0 AND SegmentID <= XPlanar.TrackCount) THEN
	_Done	 := FALSE;
	_Error	 := FALSE;
	_Busy	 := FALSE;
	_ErrorID := 0;
	ipTrack.pm.StartFromTrack(_PlanarFb, ip.Tracks[SegmentID].pm);
	HasRun := TRUE;
END_IF

Execute := THIS^;

//Heartbeat that the method is active
ExecuteWatchdog := ExecuteWatchdog + 1;
END_METHOD

END_FUNCTION_BLOCK

// Track/TaskClasses/FB_TrackReset
FUNCTION_BLOCK FB_TrackReset EXTENDS FB_TrackTask
VAR
END_VAR

METHOD Execute : I_PlanarTaskResult
IF NOT HasRun THEN
	_Done	 := FALSE;
	_Error	 := FALSE;
	_Busy	 := FALSE;
	_ErrorID := 0;
	ipTrack.pm.Reset(_PlanarFb);
	HasRun := TRUE;
END_IF

Execute := THIS^;

//Heartbeat that the method is active
ExecuteWatchdog := ExecuteWatchdog + 1;
END_METHOD

END_FUNCTION_BLOCK

// Track/FB_XPlanarTrackSegment
{attribute 'no_assign'}
{attribute 'no_explicit_call' := 'do not call this POU directly'}
FUNCTION_BLOCK FB_XPlanarTrackSegment IMPLEMENTS I_Initializable, I_Cyclic, I_XPlanarTrack
VAR
	//Planar Track 
	{attribute 'suppress_wrn_C0540'}
	_Track			: MC_PlanarTrack;
	_Definition		: ST_TrackDefinition;
	ipMcPlanarTrack : I_McPlanarTrack;

	//Track Segment Task Classes
	AppendLineToSegment	  : FB_AppendLine		 := (Track := THIS^);
	AppendPointToSegment  : FB_AppendPoint		 := (Track := THIS^);
	CloseTheLoop		  : FB_CloseLoop		 := (Track := THIS^);
	EnableTrack			  : FB_EnableTrack		 := (Track := THIS^);
	DisableTrack		  : FB_DisableTrack		 := (Track := THIS^);
	ClearTrackPoints	  : FB_ClearSegment		 := (Track := THIS^);
	AddTrackToGroup		  : FB_AddTrackToGroup	 := (Track := THIS^);
	SetStartFromTrackTask : FB_SetStartFromTrack := (Track := THIS^);
	SetEndAtTrackTask	  : FB_SetEndAtTrack	 := (Track := THIS^);
	ResetTrack			  : FB_TrackReset		 := (Track := THIS^);
	BuildTrack			  : FB_BuildTrack		 := (Track := THIS^);

	//Internal Vars
	_Initialized : BOOL;
	_Busy		 : BOOL;
	_Error		 : BOOL;
	_ErrorID	 : UDINT;
	_std		 : CDT_MCTOPLC_PLANAR_TRACK;
	_TrackLength : LREAL;
	_TrackID	 : UDINT;
	_IsStanding	 : BOOL;
	ToMCMapStatus		 : EPlcMappingStatus;
	FromMCMapStatus		 : EPlcMappingStatus;
	LinkErrMsg			 : BOOL;
END_VAR

METHOD Initialize
//Make sure track is linkted to MC3 Object
FromMCMapStatus := F_GetMappingStatus(ADR(_Track.MCTOPLC_STD), SIZEOF(_Track.MCTOPLC_STD));

IF FromMCMapStatus = EPlcMappingStatus.MS_Unmapped THEN
	IF NOT LinkErrMsg THEN
		ADSLOGDINT(ADSLOG_MSGTYPE_ERROR, 'Object not linked to MC! Track: %d', TO_DINT(_TrackId));
		LinkErrMsg := TRUE;
	END_IF
	RETURN;
END_IF
_Initialized := TRUE;
END_METHOD

{attribute 'monitoring' := 'call'}
PROPERTY Initialized : BOOL
GET
Initialized := _Initialized;
END_GET
SET
_Initialized := Initialized;
END_SET
END_PROPERTY

METHOD AddToGroup : I_PlanarTaskResult
VAR_INPUT
	PlanarGroup : REFERENCE TO MC_PlanarGroup;
END_VAR
AddToGroup := AddTrackToGroup.Execute(PlanarGroup);
END_METHOD

METHOD AppendLine : I_PlanarTaskResult
VAR_INPUT
	StartPointX : LREAL;
	StartPointY : LREAL;
	EndPointX	: LREAL;
	EndPointY	: LREAL;
END_VAR

VAR_INST
END_VAR
AppendLine := AppendLineToSegment.Execute(StartPointX,
										  StartPointY,
										  EndPointX,
										  EndPointY);
END_METHOD

METHOD AppendPoint : I_PlanarTaskResult
VAR_INPUT
	XPoint : LREAL;
	YPoint : LREAL;
END_VAR

VAR_INST
END_VAR
AppendPoint := AppendPointToSegment.Execute(XPoint, YPoint);
END_METHOD

METHOD Build : I_PlanarTaskResult
Build := BuildTrack.Execute();
END_METHOD

PROPERTY Busy : BOOL
GET
Busy := _Busy;
END_GET
END_PROPERTY

METHOD Clear : I_PlanarTaskResult
VAR_INST
	nStateReset : UINT;
END_VAR
Clear := ClearTrackPoints.Execute();
END_METHOD

METHOD CloseLoop : I_PlanarTaskResult
CloseLoop := CloseTheLoop.Execute();
END_METHOD

{attribute 'suppress_wrn_C0410'}
PROPERTY Definition : REFERENCE TO ST_TrackDefinition
GET
Definition ref= _Definition;
END_GET
END_PROPERTY

METHOD Disable : I_PlanarTaskResult
Disable := DisableTrack.Execute();
END_METHOD

{attribute 'TcRpcEnable'}
METHOD Enable : I_PlanarTaskResult
Enable := EnableTrack.Execute();
END_METHOD

PROPERTY Error : BOOL
GET
Error := _Error;
END_GET
END_PROPERTY

PROPERTY ErrorId : UDINT
GET
ErrorId := ErrorID;
END_GET
END_PROPERTY

METHOD GetTrackPositionAt : LREAL;
VAR_IN_OUT
	Position : PositionXYC;
END_VAR
GetTrackPositionAt := _Track.GetArcLengthClosestTo(Position);
END_METHOD

PROPERTY Index : UDINT
GET
Index := _TrackID;
END_GET
SET
_TrackID := Index;
END_SET
END_PROPERTY

PROPERTY IsStanding : BOOL
GET
IsStanding := _IsStanding;
END_GET
END_PROPERTY

PROPERTY MoverCount : UDINT
GET
MoverCount := _Track.MCTOPLC_STD.MoverCountOnTrack;
END_GET
END_PROPERTY

PROPERTY MovingMoverCount : UDINT
GET
MovingMoverCount := _Track.MCTOPLC_STD.MovingMoverCount;
END_GET
END_PROPERTY

{attribute 'suppress_wrn_C0410'}
PROPERTY pm : REFERENCE TO MC_PlanarTrack
GET
pm ref= _Track;
END_GET
END_PROPERTY

METHOD Reset : I_PlanarTaskResult
VAR_INPUT
END_VAR
Reset := ResetTrack.Execute();
END_METHOD

METHOD SetEndAtTrack : I_PlanarTaskResult
VAR_INPUT
	SegmentID : UDINT;
END_VAR
SetEndAtTrack := SetEndAtTrackTask.Execute(SegmentID);
END_METHOD

METHOD SetStartFromTrack : I_PlanarTaskResult
VAR_INPUT
	SegmentID : UDINT;
END_VAR
SetStartFromTrack := SetStartFromTrackTask.Execute(SegmentID);
END_METHOD

{attribute 'suppress_wrn_C0410'}
PROPERTY Status : REFERENCE TO CDT_MCTOPLC_PLANAR_TRACK
GET
Status ref= _std;
END_GET
END_PROPERTY

PROPERTY TrackLength : LREAL
GET
TrackLength := _Track.GetLength();
END_GET
END_PROPERTY

PROPERTY Utility : I_McPlanarTrack
GET
IF ipMcPlanarTrack <> 0 THEN
	Utility := ipMcPlanarTrack;
END_IF
END_GET
SET
ipMcPlanarTrack := Utility;
END_SET
END_PROPERTY

METHOD CyclicLogic
VAR
	Result : BOOL;
END_VAR
_std := _Track.MCTOPLC_STD;
EnableTrack.CyclicLogic();
DisableTrack.CyclicLogic();
AppendLineToSegment.CyclicLogic();
AppendPointToSegment.CyclicLogic();
ClearTrackPoints.CyclicLogic();
CloseTheLoop.CyclicLogic();
AddTrackToGroup.CyclicLogic();
SetStartFromTrackTask.CyclicLogic();
SetEndAtTrackTask.CyclicLogic();
ResetTrack.CyclicLogic();
BuildTrack.CyclicLogic();

_IsStanding := _std.OperationMode = Mc_Planar_Track_Operation_Mode.Standing;
END_METHOD

//FB_Init is always available implicitly and it is used primarily for initialization.
//The return value is not evaluated. For a specific influence, you can also declare the
//methods explicitly and provide additional code there with the standard initialization
//code. You can evaluate the return value.
METHOD FB_Init: BOOL
VAR_INPUT
    bInitRetains: BOOL; // TRUE: the retain variables are initialized (reset warm / reset cold)
    bInCopyCode: BOOL;  // TRUE: the instance will be copied to the copy code afterward (online change)   
END_VAR
VAR
	i	: UINT;
END_VAR
IF NOT bInCopyCode THEN
	FOR i := 1 TO Tc3_XPlanarUtility.Param_TcIoXPlanarEnvironment.MaxTracks DO
		IF ip.Tracks[i] = 0 THEN
			ip.Tracks[i] := THIS^;
			ip.Tracks[i].Index := i;
			XPlanar.TrackCount := i;
			EXIT;
		END_IF 
	END_FOR
END_IF
END_METHOD

END_FUNCTION_BLOCK

// XPlanarComponent/TaskClasses/FB_AbortSystem
FUNCTION_BLOCK FB_AbortSystem EXTENDS FB_XPlanarTaskBase
VAR
	_AbortSystem   : BOOL;
	MoversHalted   : BOOL;
	MoversDisabled : BOOL;
	TracksDisabled : BOOL;
	AbortState	   : (Init,
		HaltMovers,
		CheckMoversHalted,
		DisableMovers,
		CHeckMoversDisabled,
		DisableTracks,
		CheckTracksDisabled,
		SystemAborted);
END_VAR

METHOD CyclicLogic
VAR_INST
	WatchdogCheck : UDINT;
	i			  : UDINT;
END_VAR
CASE AbortState OF
	Init:
		IF _AbortSystem THEN
			_AbortSystem := FALSE;
			AbortState := HaltMovers;
		END_IF
		
	HaltMovers:
		FOR i := 1 TO XPlanar.MoverCount DO
			ip.Movers[i].Halt();
		END_FOR

		AbortState := CheckMoversHalted;

	CheckMoversHalted: //Monitor Halt System Feedback
		MoversHalted := TRUE;
		FOR i := 1 TO XPlanar.MoverCount DO
			IF ip.Movers[i].Status.Busy.busyMover AND (ip.Movers[i].Status.State <> Mc_Planar_State.Error) THEN
				MoversHalted := FALSE;
			END_IF
		END_FOR

		IF MoversHalted THEN
			AbortState := DisableMovers;
		END_IF

	DisableMovers: //Disable Movers
		FOR i := 1 TO XPlanar.MoverCount DO
			ip.Movers[i].Disable();
		END_FOR

		AbortState := CheckMoversDisabled;

	CheckMoversDisabled: //Check disable command feedback
		MoversDisabled := TRUE;
		FOR i := 1 TO XPlanar.MoverCount DO
			IF (ip.Movers[i].Status.State <> Mc_Planar_State.Disabled) AND (ip.Movers[i].Status.State <> Mc_Planar_State.Error) THEN
				MoversDisabled := FALSE;
			END_IF
		END_FOR

		IF MoversDisabled THEN
			AbortState := DisableTracks;
		END_IF

	DisableTracks: //Disable Tracks
		FOR i := 1 TO XPlanar.TrackCount DO
			ip.Tracks[i].Disable();
		END_FOR

		AbortState := CheckTracksDisabled;

	CheckTracksDisabled: //Monitor track disable feedback
		TracksDisabled := TRUE;
		FOR i := 1 TO XPlanar.TrackCount DO
			IF (ip.Tracks[i].Status.State <> Mc_Planar_State.Disabled) AND (ip.Tracks[i].Status.State <> Mc_Planar_State.Error) THEN
				TracksDisabled := FALSE;
			END_IF
		END_FOR

		AbortState := SystemAborted;

	SystemAborted: //Abort Complete	
		_Done	   := TRUE;
		AbortState := Init;

	999: //Error
		_Error	   := TRUE;
		AbortState := Init;
END_CASE

IF ExecuteWatchdog <> WatchdogCheck THEN
	WatchdogCheck := ExecuteWatchdog;
ELSE
	HasRun			:= FALSE;
	TaskState		:= 0;
	ExecuteWatchdog := 0;
END_IF
END_METHOD

METHOD Execute : I_PlanarTaskResult
IF NOT HasRun THEN
	_Done		 := FALSE;
	_Error		 := FALSE;
	_Busy		 := FALSE;
	_ErrorID	 := 0;
	_AbortSystem := TRUE;
	HasRun		 := TRUE;
END_IF

Execute := THIS^;

//Heartbeat that the method is active
ExecuteWatchdog := ExecuteWatchdog + 1;
END_METHOD

END_FUNCTION_BLOCK

// XPlanarComponent/TaskClasses/FB_EnableGroup
FUNCTION_BLOCK FB_EnableGroup EXTENDS FB_XPlanarTaskBase
VAR
END_VAR

METHOD Execute : I_PlanarTaskResult
IF NOT HasRun AND XPlanar.Group.MCTOPLC_STD.State = MC_PLANAR_STATE.Disabled THEN
	_Done	 := FALSE;
	_Error	 := FALSE;
	_Busy	 := FALSE;
	_ErrorID := 0;
	XPlanar.Group.Enable(_PlanarFb);
	HasRun := TRUE;
END_IF

Execute := THIS^;

//Heartbeat that the method is active
ExecuteWatchdog := ExecuteWatchdog + 1;
END_METHOD

END_FUNCTION_BLOCK

// XPlanarComponent/TaskClasses/FB_MoverIdentification
FUNCTION_BLOCK FB_MoverIdentification EXTENDS FB_XPlanarTaskBase
VAR
	_MoverIdentificationStatus : CoordinatedMoverCommStatus;
	_CoordinatedMoverComm	   : CoordinatedMoverCommCommand;
END_VAR

METHOD CyclicLogic
VAR
	i	: UDINT;
END_VAR
VAR_INST
	WatchdogCheck	: UDINT;
	RT_UpdateMovers : R_Trig;
END_VAR
IF ExecuteWatchdog <> WatchdogCheck THEN
	_MoverIdentificationStatus := XPlanar.EnvironmentTcIo.TcIoXpu(1).GetCoordMoverCommStatus();
	WatchdogCheck			   := ExecuteWatchdog;
ELSE
	HasRun := FALSE;
	ExecuteWatchdog := 0;
END_IF

THIS^.Busy	:= _MoverIdentificationStatus = CoordinatedMoverCommStatus.CommunicationInProcess;
THIS^.Done	:= _MoverIdentificationStatus = CoordinatedMoverCommStatus.CommunicationSuccessful;
THIS^.Error := _MoverIdentificationStatus = CoordinatedMoverCommStatus.CommunicationFailed;

RT_UpdateMovers(CLK := _Done);
IF RT_UpdateMovers.Q THEN
	FOR i := 1 TO XPlanar.MoverCount DO
		IF ip.Movers[i] <> 0 THEN
			ip.Movers[i].IdentifiedBTN := ip.Movers[i].Utility.GetIdentifiedMoverBtn();
		END_IF
	END_FOR
END_IF
END_METHOD

METHOD Execute : I_PlanarTaskResult
VAR_INPUT
	ReadBtnOnly	: BOOL := FALSE;
END_VAR
IF XPlanar.OperationMode = XPlanarOperationMode.Normal THEN
	IF NOT HasRun THEN
		_Done	 := FALSE;
		_Error	 := FALSE;
		_Busy	 := FALSE;
		_ErrorID := 0;
		
		IF ReadBtnOnly THEN
			_CoordinatedMoverComm := 2;
		ELSE
			_CoordinatedMoverComm := 0;
		END_IF
		
		Xplanar.EnvironmentTcIo.TcIoXpu(1).SetCoordMoverCommunicationCmd(_CoordinatedMoverComm);
		HasRun := TRUE;
	END_IF
END_IF

Execute := THIS^;

//Heartbeat that the method is active
ExecuteWatchdog := ExecuteWatchdog + 1;
END_METHOD

END_FUNCTION_BLOCK

// XPlanarComponent/TaskClasses/FB_MoverRedetection
FUNCTION_BLOCK FB_MoverRedetection EXTENDS FB_XPlanarTaskBase
VAR
	_MoverDetectionStatus : MoverDetectionStatus;
	_MoverDetectionInfo	  : ST_TcIoMoverDetectionInfos;
END_VAR

METHOD CyclicLogic
VAR_INST
	WatchdogCheck : UDINT;
	RT_UpdateInfo : R_Trig;
END_VAR
IF ExecuteWatchdog <> WatchdogCheck THEN
	_MoverDetectionStatus := XPlanar.EnvironmentTcIo.TcIoXpu(1).GetMoverDetectionStatus();
	WatchdogCheck		  := ExecuteWatchdog;
ELSE
	HasRun			:= FALSE;
	ExecuteWatchdog := 0;
END_IF

THIS^.Busy	:= _MoverDetectionStatus = MoverDetectionStatus.DetectionInProcess;
THIS^.Done	:= _MoverDetectionStatus = MoverDetectionStatus.DetectionSuccessful;
THIS^.Error := _MoverDetectionStatus = MoverDetectionStatus.NotInitialized;

RT_UpdateInfo(CLK := _Done);
IF RT_UpdateInfo.Q THEN
	_MoverDetectionInfo := XPlanar.EnvironmentTcIo.TcIoXpu(1).GetMoverDetectionInfos();
END_IF
END_METHOD

METHOD Execute : I_PlanarTaskResult
IF NOT HasRun THEN
	_Done	 := FALSE;
	_Error	 := FALSE;
	_Busy	 := FALSE;
	_ErrorID := 0;
	Xplanar.EnvironmentTcIo.TcIoXpu(1).SetStartMoverRedetection();
	HasRun := TRUE;
END_IF

Execute := THIS^;

//Heartbeat that the method is active
ExecuteWatchdog := ExecuteWatchdog + 1;
END_METHOD

PROPERTY MoverDetectionInfo : REFERENCE TO ST_TcIoMoverDetectionInfos
GET
MoverDetectionInfo ref= _MoverDetectionInfo;
END_GET
END_PROPERTY

END_FUNCTION_BLOCK

// XPlanarComponent/TaskClasses/FB_ResetGroup
FUNCTION_BLOCK FB_ResetGroup EXTENDS FB_XPlanarTaskBase
VAR
END_VAR

METHOD Execute : I_PlanarTaskResult
IF NOT HasRun AND XPlanar.Group.Error THEN
	_Done	 := FALSE;
	_Error	 := FALSE;
	_Busy	 := FALSE;
	_ErrorID := 0;
	XPlanar.Group.Reset(_PlanarFb);
	HasRun := TRUE;
END_IF

Execute := THIS^;

//Heartbeat that the method is active
ExecuteWatchdog := ExecuteWatchdog + 1;
END_METHOD

END_FUNCTION_BLOCK

// XPlanarComponent/TaskClasses/FB_ResetXPlanar
FUNCTION_BLOCK FB_ResetXPlanar EXTENDS FB_XPlanarTaskBase
VAR
	_MoverDetectionStatus : MoverDetectionStatus;
	_MoverDetectionInfo	  : ST_TcIoMoverDetectionInfos;
END_VAR

METHOD CyclicLogic
VAR_INST
	WatchdogCheck : UDINT;
END_VAR
IF ExecuteWatchdog <> WatchdogCheck THEN
	WatchdogCheck := ExecuteWatchdog;
ELSE
	HasRun			:= FALSE;
	TaskState		:= 0;
	ExecuteWatchdog := 0;
END_IF

_PlanarFb.Update();
THIS^.Busy := TaskState > 0 AND TaskState < 50;
END_METHOD

METHOD Execute : I_PlanarTaskResult
VAR_INST
	i	: UDINT;
	MoverResetResult	: I_PlanarTaskResult;
	TrackResetResult	: I_PlanarTaskResult;
END_VAR
CASE TaskState OF
	0: //Init
		i		  := 1;
		_Done	  := FALSE;
		_Error	  := FALSE;
		TaskState := TaskState + 10;

	10: //Reset Movers
		IF i <= XPlanar.MoverCount THEN
			MoverResetResult := ip.Movers[i].Reset();
			IF MoverResetResult.Done THEN
				TaskState := TaskState + 1;
			ELSIF MoverResetResult.Error THEN
				TaskState := 997;
			END_IF
		ELSE
			i		  := 1;
			TaskState := TaskState + 10;
		END_IF

	11: //Increment Index
		i		  := i + 1;
		TaskState := TaskState - 1;

	20: //Reset Track Segments
		IF i <= XPlanar.TrackCount THEN
			TrackResetResult := ip.Tracks[i].Reset();
			IF TrackResetResult.Done THEN
				TaskState := TaskState + 1;
			ELSIF TrackResetResult.Error THEN
				TaskState := 998;
			END_IF
		ELSE
			i		  := 1;
			TaskState := TaskState + 10;
		END_IF

	21: //Increment Index
		i		  := i + 1;
		TaskState := TaskState - 1;

	30: //Reset Group
		IF XPlanar.Group.Error THEN
			XPlanar.Group.Reset(_PlanarFb);
		END_IF

		TaskState := TaskState + 10;

	40: //Check Group Reset Command Feedback
		IF _PlanarFb.Done OR NOT XPlanar.Group.Error THEN
			TaskState := TaskState + 10;
		ELSIF _PlanarFb.Error THEN
			TaskState := 999;
		END_IF

	50: //Reset Complete
		_Done := TRUE;

	997: //Mover Reset Error
		_Error				:= MoverResetResult.Error;
		_ErrorID			:= MoverResetResult.ErrorID;
		_BlockingObjectInfo := MoverResetResult.BlockingObjectInfo;

	998: //Mover Reset Error
		_Error				:= TrackResetResult.Error;
		_ErrorID			:= TrackResetResult.ErrorID;
		_BlockingObjectInfo := TrackResetResult.BlockingObjectInfo;

	999: //Group Reset Error
		_Error				:= _PlanarFb.Error;
		_ErrorID			:= _PlanarFb.ErrorId;
		_BlockingObjectInfo := _PlanarFb.objectInfo;
END_CASE

Execute := THIS^;

//Heartbeat that the method is active
ExecuteWatchdog := ExecuteWatchdog + 1;
END_METHOD

END_FUNCTION_BLOCK

// XPlanarComponent/FB_Component_XPlanar
{attribute 'no_assign'}
{attribute 'no_explicit_call' := 'do not call this POU directly'}
FUNCTION_BLOCK FB_Component_XPlanar IMPLEMENTS I_XPlanarSystem, I_Cyclic, I_Initializable
VAR
	UtilityVisu : FB_XPlanarUtilityVisu;

	//System Level Tasks
	EnablePlanarGroup	: FB_EnableGroup;
	MoverDetection		: FB_MoverRedetection;
	MoverIdentification : FB_MoverIdentification;
	XPlanarReset		: FB_ResetXPlanar;
	AbortSystem			: FB_AbortSystem;
	
	//Internal Vars
	_Busy				: BOOL;
	_Error				: BOOL;
	_ErrorID			: UDINT;
	_Initialized		: BOOL;
	_OperationMode		: XPlanarOperationMode;
	_Xpu				: I_TcIoXPlanarProcessingUnit;
	_TracksInitialized	: BOOL;
	_MoverDetectionInfo : ST_TcIoMoverDetectionInfos;
	
	InitState			: (InitEnvironment,
		GetOperationMode,
		GetXPUOids,
		SetXPUInterface,
		GetPartOids,
		AssignPartOids,
		InitCurrentPart,
		NextPart,
		InitializeMovers,
		SetTrackIndex,
		GetTileCount,
		InitializeTiles,
		InitializeTracks,
		InitializeComplete,
		InitError);
END_VAR

METHOD PUBLIC CyclicLogic
VAR_INST
	i : UDINT;
END_VAR
//Update Xplanar system status
XPlanar.Environment.Update();
XPlanar.Group.Update();

//Update Movers - Must be called every cycle 
FOR i := 1 TO Param_TcIoXPlanarEnvironment.MaxMcPlanarMovers DO
	IF ip.Movers[i] <> 0 THEN
		ip.Movers[i].pm.Update();
		IF _Initialized THEN
			ip.Movers[i].CyclicLogic();
		END_IF
	ELSE
		EXIT;
	END_IF
END_FOR

//Update Tracks - Must be called every cycle 
FOR i := 1 TO Param_TcIoXPlanarEnvironment.MaxTracks DO
	IF ip.Tracks[i] <> 0 THEN
		ip.Tracks[i].pm.Update();
		IF _Initialized THEN
			ip.Tracks[i].CyclicLogic();
		END_IF
	ELSE
		EXIT;
	END_IF
END_FOR

FOR i := 1 TO SystemParameters.MAX_STATION_COUNT DO
	IF ip.Stations[i] <> 0 THEN
		ip.Stations[i].CyclicLogic();
	ELSE
		EXIT;
	END_IF
END_FOR

EnablePlanarGroup.CyclicLogic();
MoverDetection.CyclicLogic();
MoverIdentification.CyclicLogic();
XPlanarReset.CyclicLogic();
AbortSystem.CyclicLogic();

FOR i := 1 TO XPlanar.PartCount DO
	XPlanar.Parts[i].CyclicLogic();
END_FOR

//Make sure things are initialized
IF NOT _Initialized THEN
	Initialize();
	RETURN;
END_IF

//Update Station IDs
FOR i := 1 TO SystemParameters.MAX_STATION_COUNT DO
	IF ip.Stations[i] <> 0 THEN
		ip.Stations[i].ID := i;
	END_IF
END_FOR

FOR i := 1 TO XPlanar.TileCount DO
	XPlanar.Tiles[i].CyclicLogic();
END_FOR

//Update Utility Visu
UtilityVisu.Cycle();
END_METHOD

METHOD Initialize
VAR_INST
	i			   : UINT;
	SequenceState  : UDINT;
	TrackToInit	   : UDINT := 1;
	TilePosition   : ST_TcIoTilePositionOnPart;
	MoverType	   : XPlanarMoverType;
	InitPartResult : I_PlanarTaskResult;
END_VAR
_Initialized := FALSE;
CASE InitState OF
	InitEnvironment: //Init XPlanar Environment
	IF Xplanar.EnvironmentTcIo.Init(TRUE) THEN
		Xplanar.EnvironmentTcIo.Init(FALSE);
		InitState := GetOperationMode;
	ELSIF Xplanar.EnvironmentTcIo.Error THEN
		RETURN;
	END_IF

	GetOperationMode: //Get Operation Mode
		XPlanar.OperationMode := XPlanar.EnvironmentTcIo.TcIoXpu(1).GetOperationMode();
		InitState			  := GetXPUOids;

	GetXPUOids: //Get XPU OIDs
		IF XPlanar.EnvironmentTcIo.P_XpuCount > 0 THEN
			IF XPlanar.EnvironmentTcIo.GetXpuOids(TRUE) THEN
				XPlanar.EnvironmentTcIo.GetXpuOids(FALSE);
				InitState := SetXPUInterface;
			ELSIF Xplanar.EnvironmentTcIo.Error THEN
				InitState := InitError;
			END_IF;
		END_IF

	SetXPUInterface: //Set XPU Interfaces
		_Xpu					:= XPlanar.EnvironmentTcIo.TcIoXpu(1);
		UtilityVisu.Environment := XPlanar.EnvironmentTcIo;
		InitState				:= GetPartOids;

	GetPartOids: //Get Part OIDs
		XPlanar.PartCount := TO_UINT(_Xpu.GetPartCount());
		IF _Xpu.GetPartOids() THEN
			InitState := AssignPartOids;
		END_IF

	AssignPartOids: //Assign OIDs to Part Objects
		IF XPlanar.PartCount > 0 THEN
			FOR i := 1 TO XPlanar.PartCount DO
				XPlanar.Parts[i].ObjectID := _Xpu.P_PartOids[i];
			END_FOR
		END_IF

		i		  := 1;
		InitState := InitCurrentPart;

	InitCurrentPart: //Initialize Parts
		IF i > 0 AND i <= XPlanar.PartCount THEN
			InitPartResult := XPlanar.Parts[i].Initialize();
			IF InitPartResult.Done THEN
				InitState := NextPart;
			ELSIF InitPartResult.Error THEN
				InitState := InitError;
			END_IF
		ELSE
			i		  := 1;
			InitState := GetTileCount;
		END_IF

	NextPart: //Loop back for next part
		i		  := i + 1;
		InitState := InitCurrentPart;

	GetTileCount: //Get Tile Count
		XPlanar.TileCount := TO_UINT(XPlanar.EnvironmentTcIo.TcIoXpu(1).GetTileCount());
		i				  := 1;
		InitState		  := InitializeTiles;

	InitializeTiles: //Initialize Tile Objects
		FOR i := 1 TO XPlanar.TileCount DO
			XPlanar.Tiles[i].Index := i;
			XPlanar.Tiles[i].Initialize();
		END_FOR

		InitState := InitializeMovers;
	
	InitializeMovers: //Set mover index values
		FOR i := 1 TO Tc3_XPlanarUtility.Param_TcIoXPlanarEnvironment.MaxMcPlanarMovers DO
			IF ip.Movers[i] <> 0 THEN
				ip.Movers[i].Utility := _Xpu.TcIoMover(TO_UINT(i));
				ip.Movers[i].Initialize();
			ELSE
				EXIT;
			END_IF
		END_FOR
	
		XPlanar.MoverCount := _Xpu.GetMoverCount();
		InitState		   := InitializeTracks;
		
	InitializeTracks:
		FOR i := 1 TO Tc3_XPlanarUtility.Param_TcIoXPlanarEnvironment.MaxTracks DO
			IF ip.Tracks[i] <> 0 THEN
				ip.Tracks[i].Initialize();
			ELSE
				EXIT;
			END_IF
		END_FOR
		InitState := InitializeComplete;
		
	InitializeComplete: //Init Complete
		_Initialized := TRUE;

	InitError: // Init Error
		_Error	 := TRUE;
		_ErrorID := 9990;
		RETURN;
END_CASE
END_METHOD

{attribute 'monitoring' := 'call'}
PROPERTY Initialized : BOOL
GET
Initialized := _Initialized;
END_GET
SET
_Initialized := Initialized;
END_SET
END_PROPERTY

METHOD Abort : I_PlanarTaskResult
Abort := AbortSystem.Execute();
END_METHOD

METHOD AddMoversToGroup : I_PlanarTaskResult
VAR_INST
	i			   : UDINT;
	Result		   : FB_TaskResult;
	AddGroupResult : I_PlanarTaskResult;
	MoversInGroup  : BOOL;
END_VAR
MoversInGroup  := FALSE;
Result.Busy	   := TRUE;
Result.Done	   := FALSE;
Result.Error   := FALSE;
Result.ErrorID := 0;
FOR i := 1 TO XPlanar.MoverCount DO
	AddGroupResult := ip.Movers[i].AddToGroup(XPlanar.Group);
	IF AddGroupResult.Error THEN
		Result.Error   := AddGroupResult.Error;
		Result.ErrorID := AddGroupResult.ErrorID;
		Result.Busy	   := FALSE;
		EXIT;
	END_IF
END_FOR

MoversInGroup := TRUE;
FOR i := 1 TO XPlanar.MoverCount DO
	IF ip.Movers[i].Status.GroupOID = 0 THEN
		MoversInGroup := FALSE;
	END_IF
END_FOR

IF MoversInGroup THEN
	Result.Busy := FALSE;
	Result.Done := TRUE;
END_IF

AddMoversToGroup := Result;
END_METHOD

METHOD AddTracksToGroup : I_PlanarTaskResult
VAR_INST
	i			   : UDINT;
	AddGroupResult : I_PlanarTaskResult;
	Result		   : FB_TaskResult;
	TracksInGroup  : BOOL;
END_VAR
TracksInGroup  := FALSE;
Result.Busy	   := TRUE;
Result.Done	   := FALSE;
Result.Error   := FALSE;
Result.ErrorID := 0;
FOR i := 1 TO XPlanar.TrackCount DO
	AddGroupResult := ip.Tracks[i].AddToGroup(XPlanar.Group);
	IF AddGroupResult.Error THEN
		Result.Error   := AddGroupResult.Error;
		Result.ErrorID := AddGroupResult.ErrorID;
		Result.Busy	   := FALSE;
		EXIT;
	END_IF
END_FOR

TracksInGroup := TRUE;
FOR i := 1 TO XPlanar.TrackCount DO
	IF ip.Tracks[i].Status.GroupOID = 0 THEN
		TracksInGroup := FALSE;
	END_IF
END_FOR

IF TracksInGroup THEN
	Result.Busy := FALSE;
	Result.Done := TRUE;
END_IF

AddTracksToGroup := Result;
END_METHOD

METHOD DisableMovers : I_PlanarTaskResult
VAR_INST
	i			   : UDINT := 1;
	j			   : UDINT := 1;
	MoversDisabled : BOOL;
	CommandResult  : I_PlanarTaskResult;
	Result		   : FB_TaskResult;
END_VAR
Result.Done	   := FALSE;
Result.Error   := FALSE;
Result.ErrorID := 0;
IF i <= XPlanar.MoverCount THEN
	CommandResult := ip.Movers[i].Disable();
	IF CommandResult.Done THEN
		i := i + 1;
	ELSIF CommandResult.Error THEN
		_ErrorID	   := CommandResult.ErrorID;
		Result.Error   := CommandResult.Error;
		Result.ErrorID := CommandResult.ErrorID;
	END_IF
ELSE
	i := 1;
END_IF

MoversDisabled := TRUE;
FOR j := 1 TO XPlanar.MoverCount DO
	IF ip.Movers[j].Status.State = Mc_Planar_State.Enabled THEN
		MoversDisabled := FALSE;
	END_IF
END_FOR

IF MoversDisabled THEN
	Result.Done := TRUE;
END_IF

DisableMovers := Result;
END_METHOD

METHOD EnableGroup : I_PlanarTaskResult
EnableGroup := EnablePlanarGroup.Execute();
END_METHOD

METHOD EnableMovers : I_PlanarTaskResult
VAR_INST
	i			  : UDINT := 1;
	j			  : UDINT := 1;
	MoversEnabled : BOOL;
	EnableResult  : I_PlanarTaskResult;
	Result		  : FB_TaskResult;
END_VAR
Result.Done	   := FALSE;
Result.Error   := FALSE;
Result.ErrorID := 0;

IF SystemParameters.FastEnable THEN
	FOR i := 1 TO XPlanar.MoverCount DO
		ip.Movers[i].Enable();
	END_FOR
ELSE
	IF i <= XPlanar.MoverCount THEN
		IF ip.Movers[i].ActualPosition.x > 0 THEN
			EnableResult := ip.Movers[i].Enable();
			IF EnableResult.Done THEN
				i := i + 1;
			ELSIF EnableResult.Error THEN
				_ErrorID	   := EnableResult.ErrorID;
				Result.Error   := EnableResult.Error;
				Result.ErrorID := EnableResult.ErrorID;
			END_IF
		END_IF
	ELSE
		i := 1;
	END_IF
END_IF

MoversEnabled := TRUE;
FOR j := 1 TO XPlanar.MoverCount DO
	IF ip.Movers[j].Status.State <> Mc_Planar_State.Enabled THEN
		MoversEnabled := FALSE;
	ELSIF ip.Movers[j].Status.State = Mc_Planar_State.Error THEN
		Result.Error := TRUE;
		//Result.ErrorID := ip.Movers[j].Status.ErrorCode;
	END_IF
END_FOR

IF MoversEnabled THEN
	Result.Done := TRUE;
END_IF

EnableMovers := Result;
END_METHOD

METHOD EnableTracks : I_PlanarTaskResult
VAR_INST
	i			  : UDINT := 1;
	j			  : UDINT := 1;
	TracksEnabled : BOOL;
	Result		  : FB_TaskResult;
	EnableResult  : I_PlanarTaskResult;
END_VAR
Result.Done	   := FALSE;
Result.Error   := FALSE;
Result.ErrorID := 0;
IF i <= XPlanar.TrackCount THEN
	EnableResult := ip.Tracks[i].Enable();
	IF EnableResult.Done THEN
		i := i + 1;
	ELSIF EnableResult.Error THEN
		_ErrorID	   := EnableResult.ErrorID;
		Result.Error   := EnableResult.Error;
		Result.ErrorID := EnableResult.ErrorID;
	END_IF
ELSE
	i := 1;
END_IF

TracksEnabled := TRUE;
FOR j := 1 TO XPlanar.TrackCount DO
	IF ip.Tracks[j].Status.State <> Mc_Planar_State.Enabled THEN
		TracksEnabled := FALSE;
	END_IF
END_FOR

IF TracksEnabled THEN
	Result.Done := TRUE;
END_IF

EnableTracks := Result;
END_METHOD

METHOD Halt : I_PlanarTaskResult
VAR_INST
	i			  : UDINT := 1;
	j			  : UDINT := 1;
	MoversHalted  : BOOL;
	CommandResult : I_PlanarTaskResult;
	Result		  : FB_TaskResult;
END_VAR
Result.Done	   := FALSE;
Result.Error   := FALSE;
Result.ErrorID := 0;
IF i <= XPlanar.MoverCount THEN
	IF ip.Movers[i].ActualPosition.x > 0 THEN
		CommandResult := ip.Movers[i].Halt();
		IF CommandResult.Done THEN
			i := i + 1;
		ELSIF CommandResult.Error THEN
			_ErrorID	   := CommandResult.ErrorID;
			Result.Error   := CommandResult.Error;
			Result.ErrorID := CommandResult.ErrorID;
		END_IF
	END_IF
ELSE
	i := 1;
END_IF

MoversHalted := TRUE;
FOR j := 1 TO XPlanar.MoverCount DO
	IF ip.Movers[j].Busy THEN
		MoversHalted := FALSE;
	END_IF
END_FOR

IF MoversHalted THEN
	Result.Done := TRUE;
END_IF

Halt := Result;
END_METHOD

METHOD IdentifyMovers : I_PlanarTaskResult
VAR_INPUT
	ReadBtnOnly	: BOOL := TRUE;
END_VAR
IdentifyMovers := MoverIdentification.Execute(ReadBtnOnly);
END_METHOD

//! Provides basic error detection and event handling for this component
METHOD PROTECTED Monitoring
(*! @descriptionThis method is called cyclically by <c>CyclicLogic()</c>*)
VAR
	i	   : UDINT;
	Result : HRESULT;
END_VAR
//Watch for mover error
FOR i := 1 TO XPlanar.MoverCount DO
	IF ip.Movers[i].Error THEN
		_Error	 := TRUE;
		_ErrorID := ip.Movers[i].ErrorID;
		EXIT;
	END_IF
END_FOR

//Watch for Track Error
FOR i := 1 TO XPlanar.TrackCount DO
	IF ip.Tracks[i].Error THEN
		_Error := TRUE;
		_ErrorID := ip.Tracks[i].ErrorID;
		EXIT;
	END_IF
END_FOR
END_METHOD

{attribute 'suppress_wrn_C0410'}
PROPERTY MoverDetectionInfo : REFERENCE TO ST_TcIoMoverDetectionInfos
GET
MoverDetectionInfo REF= MoverDetection.MoverDetectionInfo;
END_GET
END_PROPERTY

METHOD MoverRedetect : I_PlanarTaskResult
VAR
	Result : BOOL;
END_VAR
MoverRedetect := MoverDetection.Execute();
END_METHOD

METHOD Reset : I_PlanarTaskResult
Reset := XPlanarReset.Execute();
END_METHOD

PROPERTY Utility : I_TcIoXPlanarProcessingUnit
GET
Utility := _Xpu;
END_GET
END_PROPERTY

END_FUNCTION_BLOCK

// XPlanarComponent/I_XPlanarSystem
INTERFACE I_XPlanarSystem EXTENDS I_Base

METHOD Abort : I_PlanarTaskResult
END_METHOD

METHOD AddMoversToGroup : I_PlanarTaskResult
END_METHOD

METHOD AddTracksToGroup : I_PlanarTaskResult
END_METHOD

METHOD DisableMovers : I_PlanarTaskResult
END_METHOD

METHOD EnableGroup : I_PlanarTaskResult
END_METHOD

METHOD EnableMovers : I_PlanarTaskResult
END_METHOD

METHOD EnableTracks : I_PlanarTaskResult
END_METHOD

METHOD Halt : I_PlanarTaskResult
END_METHOD

METHOD IdentifyMovers : I_PlanarTaskResult
VAR_INPUT
	ReadBtnOnly	: BOOL := FALSE;
END_VAR
END_METHOD

{attribute 'suppress_wrn_C0410'}
PROPERTY MoverDetectionInfo : REFERENCE TO ST_TcIoMoverDetectionInfos
GET
END_GET
END_PROPERTY

METHOD MoverRedetect : I_PlanarTaskResult
END_METHOD

METHOD Reset : I_PlanarTaskResult
END_METHOD

PROPERTY Utility : I_TcIoXPlanarProcessingUnit
GET
END_GET
END_PROPERTY

END_INTERFACE
